FUNCTION_BLOCK FB1
  (* Standard: 61499-2 *)
  (* Version 11-01-12, GASR *)
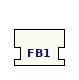
  EC_STATES
    START;
  END_STATES
END_FUNCTION_BLOCK
